FUNCTION_BLOCK Conv2Ctrl (* Basic Function Block Type *)
  (* Standard: 61499-2 *)
  (* Version 0.0, 5/8/2018, Aalto_IT, nxtControl GmbH, Template *)
  PACKAGE Main;
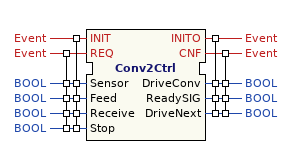
  EVENT_INPUT
    INIT WITH Sensor, Feed, Receive, Stop; (* Initialization Request *)
    REQ WITH Sensor, Feed, Receive, Stop; (* Normal Execution Request *)
  END_EVENT
  EVENT_OUTPUT
    INITO WITH DriveConv, ReadySIG, DriveNext; (* Initialization Confirm *)
    CNF WITH DriveConv, ReadySIG, DriveNext; (* Execution Confirmation *)
  END_EVENT
  VAR_INPUT
    Sensor : BOOL; (* Input event qualifier *)
    Feed : BOOL;
    Receive : BOOL;
    Stop : BOOL;
  END_VAR
  VAR_OUTPUT
    DriveConv : BOOL; (* Output event qualifier *)
    ReadySIG : BOOL;
    DriveNext : BOOL;
  END_VAR
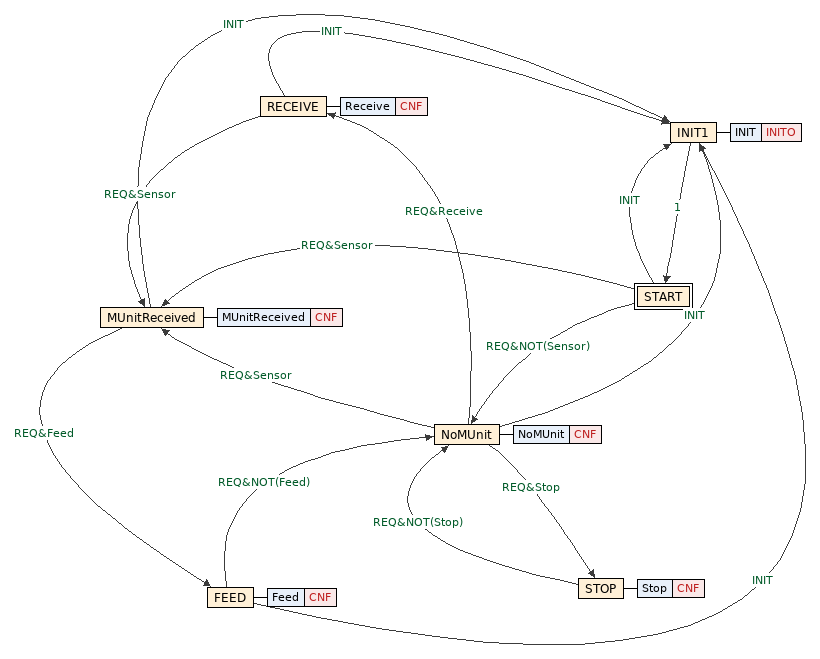
  EC_STATES
    START; (* Initial State *)
    INIT1 : INIT -> INITO; (* Initialization *)
    FEED : Feed -> CNF; (* Normal execution *)
    MUnitReceived : MUnitReceived -> CNF; (* Normal execution *)
    NoMUnit : NoMUnit -> CNF;
    RECEIVE : Receive -> CNF;
    STOP : Stop -> CNF;
  END_STATES
  EC_TRANSITIONS
    NoMUnit TO MUnitReceived := REQ&Sensor;
    MUnitReceived TO FEED := REQ&Feed;
    FEED TO NoMUnit := REQ&NOT(Feed);
    RECEIVE TO MUnitReceived := REQ&Sensor;
    NoMUnit TO RECEIVE := REQ&Receive;
    RECEIVE TO INIT1 := INIT;
    NoMUnit TO INIT1 := INIT;
    FEED TO INIT1 := INIT;
    MUnitReceived TO INIT1 := INIT;
    NoMUnit TO STOP := REQ&Stop;
    STOP TO NoMUnit := REQ&NOT(Stop);
    START TO NoMUnit := REQ&NOT(Sensor);
    INIT1 TO START := 1;
    START TO INIT1 := INIT;
    START TO MUnitReceived := REQ&Sensor;
  END_TRANSITIONS
  ALGORITHM INIT IN ST: (* Initialization algorithm *)
;
DriveConv:=0;
ReadySIG:=1;
DriveNext:=0;
  END_ALGORITHM
  ALGORITHM NoMUnit IN ST:
;
DriveConv:=0;
ReadySIG:=1;
DriveNext:=0;
  END_ALGORITHM
  ALGORITHM MUnitReceived IN ST:
;
DriveConv:=0;
ReadySIG:=0;
DriveNext:=0;
  END_ALGORITHM
  ALGORITHM Receive IN ST:
;
DriveConv:=1;
ReadySIG:=1;
DriveNext:=0;
  END_ALGORITHM
  ALGORITHM Feed IN ST:
;
DriveConv:=1;
ReadySIG:=0;
DriveNext:=1;
  END_ALGORITHM
  ALGORITHM Stop IN ST:
;
DriveConv:=0;
ReadySIG:=0;
DriveNext:=0;
  END_ALGORITHM
END_FUNCTION_BLOCK
